Staubli VAL3: printDebug.pgx

public program printDebug(string x_sDebugMessage (dimensions=1), bool x_bStamp (dimensions=1))
begin
  // Copyright (c) 2021, Institute for Factory Automation and Production Systems (FAPS)
  //
  // Licensed under the Apache License, Version 2.0 (the "License");
  // you may not use this file except in compliance with the License.
  // You may obtain a copy of the License at
  //
  //     http://www.apache.org/licenses/LICENSE-2.0
  //
  // Unless required by applicable law or agreed to in writing, software
  // distributed under the License is distributed on an "AS IS" BASIS,
  // WITHOUT WARRANTIES OR CONDITIONS OF ANY KIND, either express or implied.
  // See the License for the specific language governing permissions and
  // limitations under the License.


  // check whether cursor is at last line (keys line)
  if (nDebugCursor==13)
    // erase line before printing the message
    put(scDebug,"                                        ")
    gotoxy(scDebug,0,13)
  endIf

  // print message
  if (x_bStamp)
    // print timestamp
    //put(scDebug,getDate("%H:%M:%S"))
    put(scDebug, "[" + toString(".3", clock()) + "] ")
  // else
    // put(scDebug,"  ")
  endIf
  putln(scDebug,x_sDebugMessage)
  nDebugCursor=sel(nDebugCursor==13,13,nDebugCursor+1)

  // update keys line if necessary
  if (nDebugCursor==13)
    gotoxy(scDebug,0,13)
    put(scDebug,"BACK")
    gotoxy(scDebug,16,13)
    put(scDebug,"CLS")
    gotoxy(scDebug,31,13)
    put(scDebug,"-")
    gotoxy(scDebug,36,13)
    put(scDebug,"+")
    gotoxy(scDebug,0,13)
  endIf
end
